{library PUBLIC}
TYPE GANTRY_STATUS :
(
	GANTRY_STATUS_NOT_ENABLED:=-1,					(* En signal is false or block is not enabled *)
	GANTRY_STATUS_NOT_READY:=0,						(* NOT ready *)
	GANTRY_STATUS_READY:=1, 							(* Auto run OK *)
	GANTRY_STATUS_INIT_MOVE:=2, 						(* Init of accelerations speeds etc *)
	GANTRY_STATUS_START_MOVE:=3,					(* Start transportation *)
	GANTRY_STATUS_MOVE_TO_STATION:=4,				(* Robot in motion *)
	GANTRY_STATUS_WAIT_CLEAR_ORDER:=5,			(* Wait until order is cleared *)
	GANTRY_STATUS_WAIT_FOR_ORDER:=6,				(* Wait for a pick or leave order *)
	GANTRY_STATUS_ORDER_ERROR:=7,				(* Error in pick or leave order *)
	GANTRY_STATUS_MOVE_TO_PICK:=8,					(* Robot picks pallet *)
	GANTRY_STATUS_WAIT_FOR_LEAVE_ORDER:=9,	(* Wait for leave order *)
	GANTRY_STATUS_ORDER_LEAVE_ERROR:=10,		(* Error in leave order *)
	GANTRY_STATUS_MOVE_TO_LEAVE:=11 				(* Robot leave pallet *)
);
END_TYPE
//  GANTRY_STATUS_NOT_ENABLED = '-1'

(* stored: Version 1.1.0.1, ProductVersion 3.1.4024.2
   EnumerationTextList GANTRY_STATUS: Id {de3744c9-a96b-4d81-89e9-44c85adf7606} *)
